// TIA Portal V19 export
DATA_BLOCK "InstLAF_MemCardDiag"   // DB126
AUTHOR : Siemens Digital Industries
FAMILY : LAF
VERSION : 1.2
// stored: AssignedProDiagFB ProDiag, InstanceOfName LAF_MemCardDiag, InstanceOfType FB
"LAF_MemCardDiag"
   // VAR_INPUT
   //    plantIdentifier { ExternalAccessible := 'False'; ExternalVisible := 'False'; ExternalWritable := 'False'} : WString[24];
   //    textListId { ExternalAccessible := 'False'; ExternalVisible := 'False'; ExternalWritable := 'False'} : Int;
   //    firstCycle { ExternalAccessible := 'False'; ExternalVisible := 'False'; ExternalWritable := 'False'} : Bool;
   //    readInfoMemCard { ExternalAccessible := 'False'; ExternalVisible := 'False'; ExternalWritable := 'False'} : Bool;
   //    hideAlarmMask { ExternalAccessible := 'False'; ExternalVisible := 'False'; ExternalWritable := 'False'} : Byte;
   // END_VAR
   // VAR_OUTPUT
   //    generalAlarm { ExternalAccessible := 'False'; ExternalVisible := 'False'; ExternalWritable := 'False'} : Bool;
   //    generalWarn { ExternalAccessible := 'False'; ExternalVisible := 'False'; ExternalWritable := 'False'} : Bool;
   //    generalInfo { ExternalAccessible := 'False'; ExternalVisible := 'False'; ExternalWritable := 'False'} : Bool;
   // END_VAR
   // VAR_IN_OUT
   //    diagHmi : "LAF_typeMemCardDiag";
   // END_VAR
   // VAR
   //    statMessages { ExternalAccessible := 'False'; ExternalVisible := 'False'; ExternalWritable := 'False'} : "LAF_typeMemCardMessages";
   //    statHideMessages { ExternalAccessible := 'False'; ExternalVisible := 'False'; ExternalWritable := 'False'} : "LAF_typeMemCardMessages";
   //    statStep { ExternalAccessible := 'False'; ExternalVisible := 'False'; ExternalWritable := 'False'} : Array[0..3] of Bool;
   //    statRisEdgeStep0 { ExternalAccessible := 'False'; ExternalVisible := 'False'; ExternalWritable := 'False'} : Bool;
   //    statRisEdgeStep1 { ExternalAccessible := 'False'; ExternalVisible := 'False'; ExternalWritable := 'False'} : Bool;
   //    statAlarmNo { ExternalAccessible := 'False'; ExternalVisible := 'False'; ExternalWritable := 'False'} : UInt;
   //    statWarnNo { ExternalAccessible := 'False'; ExternalVisible := 'False'; ExternalWritable := 'False'} : UInt;
   //    statInfoNo { ExternalAccessible := 'False'; ExternalVisible := 'False'; ExternalWritable := 'False'} : UInt;
   //    instGetInfoMode0 { ExternalAccessible := 'False'; ExternalVisible := 'False'; ExternalWritable := 'False'} : GetSMCinfo;
   //    instGetInfoMode1 { ExternalAccessible := 'False'; ExternalVisible := 'False'; ExternalWritable := 'False'} : GetSMCinfo;
   //    instGetInfoMode2 { ExternalAccessible := 'False'; ExternalVisible := 'False'; ExternalWritable := 'False'} : GetSMCinfo;
   //    instGetInfoMode3 { ExternalAccessible := 'False'; ExternalVisible := 'False'; ExternalWritable := 'False'} : GetSMCinfo;
   // END_VAR
BEGIN
END_DATA_BLOCK
